(* CODESYS project NativeMQTT-Node-RED-Publish.ecp
   Company: WAGO
   Title: WagoAppCloud_CostumerProtocol
   Description: Example for the Cloud Conectivity using MQTT with the own customer data strucure
   Author: wago / u014791
   Version: 1.0.0.0

Project tree, tasks and I/O mapping:
  PFC : 750-8212 PFC200 2ETH RS, WAGO, order no. 0750-8212, version 5.13.2.32
    application Application
      libraries: WagoAppString, 1.6.3.1 (WAGO); WagoAppJSON, 1.0.2.0 (WAGO); WagoAppCloud, 1.3.0.8 (WAGO)
      task Task (cyclic, interval t#10ms, priority 14) calls PLC_PRG
      program Status_NativeMQTT [ST]
      data type ByteToString
      program PLC_PRG [ST]
      program PRG_Build_JSON [ST]
      program PRG_NativeMQTT [ST]: ACT_GetData
    Kbus : Kbus, WAGO, version 1.4.0.2
        unmapped channels: K-BUS diagnostics
    MODBUS
      MODBUS : MODBUS, WAGO, order no. n/a, version 1.1.1.15
    Serial
      COM1 : COM1, WAGO, version 0.0.0.19
    Common.PCI
*)

// PFC/Application/ByteToString
TYPE ByteToString :
UNION
	abData: ARRAY[0..99] OF BYTE;
	abDataBig: ARRAY[0..999] OF BYTE;
	sData: STRING(100);
END_UNION
END_TYPE

// PFC/Application/PLC_PRG
PROGRAM PLC_PRG
VAR
END_VAR

PRG_Build_JSON();
PRG_NativeMQTT();		
Status_NativeMQTT();

END_PROGRAM

// PFC/Application/PRG_Build_JSON
PROGRAM PRG_Build_JSON
VAR
	oFb_JSON: WagoAppJSON.Fb_JSON_Writer_01;
	MyTemplateString :STRING(1000) := 
					'{"Temperature": "#Parameter","Voltage": "#Parameter","Counting Number": "#Parameter"}';
					// "#Parameter" will be replaced with the array value starting by array index"0" to "2"			
	asMyValueArray	: ARRAY [0..2] OF STRING;
	sOutput			: STRING(JSON_MAX_STRING);
	bMyValue		: BYTE := 1;
END_VAR

VAR_INPUT
	xTrigger_Update_Payload: BOOL := TRUE;
END_VAR

//Values for "#Parameter"
asMyValueArray[0]:= TO_STRING(bMyValue/10.0);
asMyValueArray[1]:= TO_STRING(bMyValue*2.3/327.6);
asMyValueArray[2]:= TO_STRING(bMyValue);
bMyValue:=bMyValue+1;


oFb_JSON(
	sJSON_BaseFrame:=MyTemplateString , 
	aParameterValues:= asMyValueArray, 
	xTrigger:= xTrigger_Update_Payload, 
	sOutput:=sOutput );

END_PROGRAM

// PFC/Application/PRG_NativeMQTT
PROGRAM PRG_NativeMQTT
VAR
	oFbPublishNativeMQTT	: WagoAppCloud.FbPublishMQTT;
	oFbStatusNativeMQTT		: WagoAppCloud.FbStatus_NativeMQTT;
	MyString				: STRING(JSON_MAX_STRING);
	dwBytesCount			: UDINT;
	abBuffer				: ARRAY[0..255] OF BYTE;
	xTrigger_Publish		: BOOL := TRUE;
	xBusy_Publish			: BOOL;
	xError_Publish			: BOOL;
	oStatus_Publish			: FbResult;
	xError_Status_MQTT		: BOOL;
	xCloudConnected			: BOOL;
	rCacheFillLevel			: REAL;
	uliOutgoingDataBlocks	: ULINT;
	oTON: Standard.TON;
	abPayloadData			: ARRAY[0..99] OF BYTE;
	xBusySub				: BOOL;
	xErrorSub				: BOOL;
	oStatusSub				: WagoAppCloud.WagoSysErrorBase.FbResult;
	xDataRxSub				: BOOL;
	dwRxNBytesSub			: DWORD;
	xDataTruncatedSub		: BOOL;
	sReceivedTopic			: STRING(255);
	oFbSubscribeNativeMQTT	: WagoAppCloud.FbSubscribeMQTT;
	oFbSubscribeNativeMQTT2 : WagoAppCloud.FbSubscribeMQTT;
	MyB2S					: ByteToString;
	sValueFromX				: STRING(100);
	
	oFbGetJSONData			: WagoAppJSON.Fb_JSON_ParseAndModify;
	oFbGetJSONData2			: WagoAppJSON.Fb_JSON_ParseAndModify;
	xTrigger_ParseData		: BOOL;
	oStatusJSONParse		: WagoAppJSON.WagoSysErrorBase.FbResult;
	xErrorJSONParse			: BOOL;
	xDoneJSONParse			: BOOL;
	diTokenJSONParse		: DINT;
	oFbJSONValue			: WagoAppJSON.Fb_JSON_ParseAndModify;
	xTrigger_GetData		: BOOL;
	sPathToValue			: STRING(SIZE_JSON_POINTER) := '/';
	typValue					: WagoAppJSON.typJSON_Pointer;

	sSubTopic: STRING(255) := 'training/nodered/myvalue';
	xSubscribe: BOOL := TRUE;
	xSubscribe2: BOOL;
	sSubTopic2: STRING(255) := 'topic';
	abPayloadData2: ARRAY [0..999] OF BYTE;
	xBusySub2: BOOL;
	xErrorSub2: BOOL;
	oStatusSub2: WagoAppCloud.WagoSysErrorBase.FbResult;
	xDataRxSub2: BOOL;
	xDataTruncatedSub2: BOOL;
	sReceivedTopic2: STRING(255);
	MyB2S_2: ByteToString;
	sValueFromX2: STRING(100);
	oStatusJSONParse2: WagoAppJSON.WagoSysErrorBase.FbResult;
	xErrorJSONParse2: BOOL;
	xDoneJSONParse2: BOOL;
	diTokenJSONParse2: DINT;
	xTrigger_ParseData2: BOOL;
	sPathToValue2: STRING(SIZE_JSON_POINTER) := '/0/level';
	xTrigger_GetData2: BOOL;
	typValue2: WagoAppJSON.typJSON_Pointer;
END_VAR

oTON(IN:=NOT oTON.Q , PT:= T#1S);
IF oTON.Q THEN
	xTrigger_Publish:=TRUE;
	PRG_Build_JSON.xTrigger_Update_Payload:=TRUE;
	xTrigger_ParseData:=TRUE;
END_IF

MyString := PRG_Build_JSON.sOutput;
dwBytesCount := Length(MyString);
MemCopy(pDest := ADR(abBuffer), pSource := ADR(MyString), udiSize := dwBytesCount);

oFbPublishNativeMQTT(
	sTopic:='training/pfc/data' ,  //--> https://thingsboard.io/docs/reference/mqtt-api/
	eQualityOfService:= eQualityOfService.QoS1, 
	xRetain:= , 
	dwSize:= dwBytesCount, 
	aData:= abBuffer, 
	xTrigger:= xTrigger_Publish, 
	xBusy=> xBusy_Publish , 
	xError=> xError_Publish, 
	oStatus=> oStatus_Publish);

ACT_GetData();



oFbStatusNativeMQTT(
	xEnabled:= TRUE, 
	xError=> xError_Status_MQTT, 
	xCloudConnected=> xCloudConnected, 
	rCacheFillLevel=> rCacheFillLevel, 
	uliOutgoingDataBlocks=> uliOutgoingDataBlocks);

ACTION ACT_GetData:
//-------------------------Singele Value Topic----------------------------------------------------

oFbSubscribeNativeMQTT(
	xSubscribe:=xSubscribe , 
	sTopic:= sSubTopic, 
	eQoS:= eQualityOfService.QoS1, 
	aPayloadData:= abPayloadData, 
	xBusy=> xBusySub , 
	xError=> xErrorSub, 
	oStatus=> oStatusSub, 
	xDataReceived=> xDataRxSub, 
	dwRxNBytes=> dwRxNBytesSub, 
	xDataTruncated=>xDataTruncatedSub , 
	sReceivedTopic=>sReceivedTopic );
	
	MyB2S.abData:=abPayloadData;
	sValueFromX:=MyB2S.sData;
	
(*oFbGetJSONData(
	pData:= ADR(sValueFromX) , 
	udiSizeData:= SIZEOF(sValueFromX), 
	oStatus=> oStatusJSONParse, 
	xError=> xErrorJSONParse, 
	xDone=>xDoneJSONParse , 
	diToken=> diTokenJSONParse, 
	xTrigger:= xTrigger_ParseData);

typValue:=oFbGetJSONData.GetValueByPath(sPointer:=sPathToValue , xTrigger:=xTrigger_GetData );
typValue.sValue;	
*)
//---------------------------Object Topic---------------------------------------------------

oFbSubscribeNativeMQTT2(
	xSubscribe:=xSubscribe2 , 
	sTopic:= sSubTopic2, 
	eQoS:= eQualityOfService.QoS1, 
	aPayloadData:= abPayloadData2, 
	xBusy=> xBusySub2 , 
	xError=> xErrorSub2, 
	oStatus=> oStatusSub2, 
	xDataReceived=> xDataRxSub2, 
	dwRxNBytes=> dwRxNBytesSub, 
	xDataTruncated=>xDataTruncatedSub2 , 
	sReceivedTopic=>sReceivedTopic2 );
	
	MyB2S_2.abDataBig:=abPayloadData2;
	sValueFromX2:=MyB2S_2.sData;
	
oFbGetJSONData2(
	pData:= ADR(sValueFromX2) , 
	udiSizeData:= SIZEOF(sValueFromX2), 
	oStatus=> oStatusJSONParse2, 
	xError=> xErrorJSONParse2, 
	xDone=>xDoneJSONParse2 , 
	diToken=> diTokenJSONParse2, 
	xTrigger:= xTrigger_ParseData2);

typValue2:=oFbGetJSONData2.GetValueByPath(sPointer:=sPathToValue2 , xTrigger:=xTrigger_GetData2 );
typValue2.sValue;
END_ACTION

END_PROGRAM

// PFC/Application/Status_NativeMQTT
// Purpose of the example program: Check status of Native MQTT
PROGRAM Status_NativeMQTT
VAR
	oFbStatus 			: WagoAppCloud.FbStatus_NativeMQTT;
	xMyError			: BOOL := FALSE;
	xConnectedToMyCloud	: BOOL := FALSE;
	rMyFillLevel		: REAL := 0;
	uliMyOutgoingBlocks	: ULINT := 0;
END_VAR

// Will detect new values every 5 seconds
oFbStatus(xEnabled := TRUE,
		   xError => xMyError,
		   xCloudConnected => xConnectedToMyCloud,			// Will be FALSE after network timeout occured 
		   rCacheFillLevel => rMyFillLevel,					// Increasing value indicates bad network or overload
		   uliOutgoingDataBlocks => uliMyOutgoingBlocks);  	// Only for QoS 1 and 2. Increasing value indicates bad network or overload

END_PROGRAM
